# B&R Automation Studio project NAELD004C00R10L518F00 (part 20)

#### InputRef.var - Change By Project
```iecst
(*2019-03-25*)
(**)
(*Configuration*)
VAR
	p_eAct : REFERENCE TO UDINT;
	p_bOpsRun : REFERENCE TO BOOL;
END_VAR
(**)
VAR
	p_eStartupStat : REFERENCE TO eStartupAction;
	p_eStartupStatus : REFERENCE TO eFBStatus;
	p_sStartupStatTxt : REFERENCE TO STRING[200];
	p_eStartupStep : REFERENCE TO eStartupStep;
	p_sStartupStepTxt : REFERENCE TO STRING[80];
	p_bStartupGetConfigDone : REFERENCE TO BOOL;
	p_bStartupMismatchSetConfigDone : REFERENCE TO BOOL;
	p_bStartupUISettingsLoadDone : REFERENCE TO BOOL;
	p_bStartupRun : REFERENCE TO BOOL;
END_VAR
(**)
VAR
	p_eHWInfoStat : REFERENCE TO eHWInfoAction;
	p_eHWInfoStatus : REFERENCE TO eFBStatus;
	p_sHWInfoStatTxt : REFERENCE TO STRING[200];
	p_sHWInfoIPAddr : REFERENCE TO STRING[15];
	p_sHWInfoSubnetMask : REFERENCE TO STRING[15];
	p_udiHWInfoEthMode : REFERENCE TO UDINT;
END_VAR
(**)
VAR
	p_eTLBuzStat : REFERENCE TO eTLBuzAction;
	p_eTLBuzStatus : REFERENCE TO eFBStatus;
	p_sTLBuzStatTxt : REFERENCE TO STRING[200];
END_VAR
(**)
VAR
	p_tyAlarmCurrList : REFERENCE TO ARRAY[1..c_udiAlarmCurrMax] OF tyAlarmCurr;
	p_tyAlarmRcyList : REFERENCE TO ARRAY[1..c_udiAlarmCurrMax] OF UDINT;
	p_tyAlarmHistoryList : REFERENCE TO ARRAY[1..c_udiAlarmHistoryMax] OF STRING[200];
	p_bAlarmWarning : REFERENCE TO BOOL;
	p_bAlarmErr : REFERENCE TO BOOL;
	p_bAlarmInfo : REFERENCE TO BOOL;
	p_bAlarmInfoLF : REFERENCE TO BOOL;
	p_sAlarmInfoMsg : REFERENCE TO STRING[200];
END_VAR
(**)
VAR
	p_eRstErrStat : REFERENCE TO eRstErrAction;
	p_eRstErrStatus : REFERENCE TO eFBStatus;
	p_sRstErrStatTxt : REFERENCE TO STRING[200];
END_VAR
(**)
VAR
	p_eProdRcpStat : REFERENCE TO eProdRcpAction;
	p_eProdRcpStatus : REFERENCE TO eFBStatus;
	p_sProdRcpStatTxt : REFERENCE TO STRING[200];
	p_tyProdRcpFilterList : REFERENCE TO ARRAY[1..c_udiProdRcpMax] OF tyProdRcpParam;
	p_tyProdRcpSortedList : REFERENCE TO ARRAY[1..c_udiProdRcpMax] OF tyProdRcpParam;
	p_tyProdRcpCurrList : REFERENCE TO ARRAY[1..c_udiProdRcpMax] OF tyProdRcpParam;
	p_tyProdRcpCurrRcp0 : REFERENCE TO tyProdRcpParam;
	p_tyProdRcpCurrRcp1 : REFERENCE TO tyProdRcpParam;
	p_tyProdRcpCurrRcp2 : REFERENCE TO tyProdRcpParam;
	p_tyProdRcpInfoOut : REFERENCE TO tyProdRcpParam;
	p_bProdRcpNmEmpty : REFERENCE TO BOOL;
	p_bProdRcpListFull : REFERENCE TO BOOL;
	p_bProdRcpNmNotExist : REFERENCE TO BOOL;
END_VAR
(**)
VAR
	p_eMpProdRcpStat : REFERENCE TO eMpProdRcpAction;
	p_eMpProdRcpStatus : REFERENCE TO eFBStatus;
END_VAR
(**)
VAR
	p_eMagRcpStat : REFERENCE TO eMagRcpAction;
	p_eMagRcpStatus : REFERENCE TO eFBStatus;
	p_sMagRcpStatTxt : REFERENCE TO STRING[200];
	p_tyMagRcpFilterList : REFERENCE TO ARRAY[1..c_udiMagRcpMax] OF tyMagRcpParam;
	p_tyMagRcpSortedList : REFERENCE TO ARRAY[1..c_udiProdRcpMax] OF tyMagRcpParam;
	p_tyMagRcpCurrList : REFERENCE TO ARRAY[1..c_udiMagRcpMax] OF tyMagRcpParam;
	p_tyMagRcpInfoOut : REFERENCE TO tyMagRcpParam;
	p_tyMagRcpCurrRcp : REFERENCE TO tyMagRcpParam;
	p_bMagRcpNmEmpty : REFERENCE TO BOOL;
	p_bMagRcpListFull : REFERENCE TO BOOL;
	p_bMagRcpNmNotExist : REFERENCE TO BOOL;
END_VAR
(**)
VAR
	p_eMagRcpStat1 : REFERENCE TO eMagRcpAction;
	p_eMagRcpStatus1 : REFERENCE TO eFBStatus;
	p_sMagRcpStatTxt1 : REFERENCE TO STRING[200];
	p_tyMagRcpFilterList1 : REFERENCE TO ARRAY[1..c_udiMagRcpMax] OF tyMagRcpParam;
	p_tyMagRcpSortedList1 : REFERENCE TO ARRAY[1..c_udiProdRcpMax] OF tyMagRcpParam;
	p_tyMagRcpCurrList1 : REFERENCE TO ARRAY[1..c_udiMagRcpMax] OF tyMagRcpParam;
	p_tyMagRcpInfoOut1 : REFERENCE TO tyMagRcpParam;
	p_tyMagRcpCurrRcp1 : REFERENCE TO tyMagRcpParam;
	p_bMagRcpNmEmpty1 : REFERENCE TO BOOL;
	p_bMagRcpListFull1 : REFERENCE TO BOOL;
	p_bMagRcpNmNotExist1 : REFERENCE TO BOOL;
	p_diMagRcp1TravPos : REFERENCE TO DINT;
	p_diMagRcp2TravPos : REFERENCE TO DINT;
	p_diMagRcp3TravPos : REFERENCE TO DINT;
END_VAR
(**)
VAR
	p_eMcParamStat : REFERENCE TO eMcParamAction;
	p_eMcParamStatus : REFERENCE TO eFBStatus;
	p_sMcParamStatTxt : REFERENCE TO STRING[200];
	p_tyMcParamCurr : REFERENCE TO tyMcParam;
END_VAR
(**)
VAR
	p_tyNtParamCurr : REFERENCE TO tyNtParam;
END_VAR
(**)
VAR
	p_eUsrMgmtStat : REFERENCE TO eUsrMgmtAction;
	p_eUsrMgmtStatus : REFERENCE TO eFBStatus;
	p_sUsrMgmtStatTxt : REFERENCE TO STRING[200];
	p_tyUsrMgmtCurrUsr : REFERENCE TO tyUsrMgmtParam;
	p_tyUsrMgmtCurrAccessRgt : REFERENCE TO tyUsrMgmtAccessRight;
	p_tyUsrMgmtAllList : REFERENCE TO ARRAY[1..c_udiUsrMgmtMax] OF tyUsrMgmtParam;
	p_tyUsrMgmtLv2List : REFERENCE TO ARRAY[1..c_udiUsrMgmtMax] OF tyUsrMgmtParam;
	p_tyUsrMgmtLv3List : REFERENCE TO ARRAY[1..c_udiUsrMgmtMax] OF tyUsrMgmtParam;
	p_tyUsrMgmtAdminList : REFERENCE TO ARRAY[1..c_udiUsrMgmtMax] OF tyUsrMgmtParam;
	p_bUsrMgmtNmEmpty : REFERENCE TO BOOL;
	p_bUsrMgmtListFull : REFERENCE TO BOOL;
	p_bUsrMgmtNmExist : REFERENCE TO BOOL;
	p_bUsrMgmtNmNotExist : REFERENCE TO BOOL;
	p_bUsrMgmtLastAdmin : REFERENCE TO BOOL;
	p_bUsrMgmtLoginSuccess : REFERENCE TO BOOL;
	p_bUsrMgmtPwMismatch : REFERENCE TO BOOL;
	p_bUsrMgmtUnableDelete : REFERENCE TO BOOL;
	p_tyUsrMgmtFullData : REFERENCE TO tyUsrMgmtFullDat;
END_VAR
(**)
VAR
	p_eBuffer1Stat : REFERENCE TO eBufferAction;
	p_eBuffer1Status : REFERENCE TO eFBStatus;
	p_sBuffer1StatTxt : REFERENCE TO STRING[200];
	p_tyBuffer1DispBffr : REFERENCE TO tyDispBffr;
	p_tyBuffer1BffrStat : REFERENCE TO tyBffrStat;
	p_bBuffer1MagPresent : REFERENCE TO BOOL;
	p_bBuffer1MagRemoved : REFERENCE TO BOOL;
END_VAR
(**)
VAR
	p_eBuffer2Stat : REFERENCE TO eBufferAction;
	p_eBuffer2Status : REFERENCE TO eFBStatus;
	p_sBuffer2StatTxt : REFERENCE TO STRING[200];
	p_tyBuffer2DispBffr : REFERENCE TO tyDispBffr;
	p_tyBuffer2BffrStat : REFERENCE TO tyBffrStat;
	p_bBuffer2MagPresent : REFERENCE TO BOOL;
	p_bBuffer2MagRemoved : REFERENCE TO BOOL;
END_VAR
(**)
VAR
	p_eBuffer3Stat : REFERENCE TO eBufferAction;
	p_eBuffer3Status : REFERENCE TO eFBStatus;
	p_sBuffer3StatTxt : REFERENCE TO STRING[200];
	p_tyBuffer3DispBffr : REFERENCE TO tyDispBffr;
	p_tyBuffer3BffrStat : REFERENCE TO tyBffrStat;
	p_bBuffer3MagPresent : REFERENCE TO BOOL;
	p_bBuffer3MagRemoved : REFERENCE TO BOOL;
END_VAR
(**)
VAR
	p_eBuffer4Stat : REFERENCE TO eBufferAction;
	p_eBuffer4Status : REFERENCE TO eFBStatus;
	p_sBuffer4StatTxt : REFERENCE TO STRING[200];
	p_tyBuffer4DispBffr : REFERENCE TO tyDispBffr;
	p_tyBuffer4BffrStat : REFERENCE TO tyBffrStat;
	p_bBuffer4MagPresent : REFERENCE TO BOOL;
	p_bBuffer4MagRemoved : REFERENCE TO BOOL;
END_VAR
(**)
VAR
	p_eDSSMEMAAStat : REFERENCE TO eSMEMAAction;
	p_eDSSMEMAAStatus : REFERENCE TO eFBStatus;
	p_sDSSMEMAAStatTxt : REFERENCE TO STRING[200];
	p_bDSSMEMAAUSRdy : REFERENCE TO BOOL;
	p_bDSSMEMAAUSGdBrdRdy : REFERENCE TO BOOL;
	p_bDSSMEMAADSRdy : REFERENCE TO BOOL;
END_VAR
(**)
VAR
	p_eDSSMEMABStat : REFERENCE TO eSMEMAAction;
	p_eDSSMEMABStatus : REFERENCE TO eFBStatus;
	p_sDSSMEMABStatTxt : REFERENCE TO STRING[200];
	p_bDSSMEMABUSRdy : REFERENCE TO BOOL;
	p_bDSSMEMABUSGdBrdRdy : REFERENCE TO BOOL;
	p_bDSSMEMABDSRdy : REFERENCE TO BOOL;
END_VAR
(**)
VAR
	p_eInShutterStat : REFERENCE TO ePneuAction;
	p_eInShutterStatus : REFERENCE TO eFBStatus;
	p_sInShutterStatTxt : REFERENCE TO STRING[200];
	p_bInShutterExtCtrl : REFERENCE TO BOOL;
	p_bInShutterRetCtrl : REFERENCE TO BOOL;
	p_bInShutterTwoCtrlOut : REFERENCE TO BOOL;
	p_bInShutterExtended : REFERENCE TO BOOL;
	p_bInShutterRetracted : REFERENCE TO BOOL;
END_VAR
(**)
VAR
	p_eInShutterStat2 : REFERENCE TO ePneuAction;
	p_eInShutterStatus2 : REFERENCE TO eFBStatus;
	p_sInShutterStatTxt2 : REFERENCE TO STRING[200];
	p_bInShutterExtCtrl2 : REFERENCE TO BOOL;
	p_bInShutterRetCtrl2 : REFERENCE TO BOOL;
	p_bInShutterTwoCtrlOut2 : REFERENCE TO BOOL;
	p_bInShutterExtended2 : REFERENCE TO BOOL;
	p_bInShutterRetracted2 : REFERENCE TO BOOL;
END_VAR
(**)
VAR
	p_eInShutterStat3 : REFERENCE TO ePneuAction;
	p_eInShutterStatus3 : REFERENCE TO eFBStatus;
	p_sInShutterStatTxt3 : REFERENCE TO STRING[200];
	p_bInShutterExtCtrl3 : REFERENCE TO BOOL;
	p_bInShutterRetCtrl3 : REFERENCE TO BOOL;
	p_bInShutterTwoCtrlOut3 : REFERENCE TO BOOL;
	p_bInShutterExtended3 : REFERENCE TO BOOL;
	p_bInShutterRetracted3 : REFERENCE TO BOOL;
END_VAR
(**)
VAR
	p_eOutShutterStat : REFERENCE TO ePneuAction;
	p_eOutShutterStatus : REFERENCE TO eFBStatus;
	p_sOutShutterStatTxt : REFERENCE TO STRING[200];
	p_bOutShutterExtCtrl : REFERENCE TO BOOL;
	p_bOutShutterRetCtrl : REFERENCE TO BOOL;
	p_bOutShutterTwoCtrlOut : REFERENCE TO BOOL;
	p_bOutShutterExtended : REFERENCE TO BOOL;
	p_bOutShutterRetracted : REFERENCE TO BOOL;
END_VAR
(**)
VAR
	p_eOutShutterStat2 : REFERENCE TO ePneuAction;
	p_eOutShutterStatus2 : REFERENCE TO eFBStatus;
	p_sOutShutterStatTxt2 : REFERENCE TO STRING[200];
	p_bOutShutterExtCtrl2 : REFERENCE TO BOOL;
	p_bOutShutterRetCtrl2 : REFERENCE TO BOOL;
	p_bOutShutterTwoCtrlOut2 : REFERENCE TO BOOL;
	p_bOutShutterExtended2 : REFERENCE TO BOOL;
	p_bOutShutterRetracted2 : REFERENCE TO BOOL;
END_VAR
(**)
VAR
	p_eSelClamp1Stat : REFERENCE TO ePneuAction;
	p_eSelClamp1Status : REFERENCE TO eFBStatus;
	p_sSelClamp1StatTxt : REFERENCE TO STRING[200];
	p_bSelClamp1ExtCtrl : REFERENCE TO BOOL;
	p_bSelClamp1RetCtrl : REFERENCE TO BOOL;
	p_bSelClamp1TwoCtrlOut : REFERENCE TO BOOL;
	p_bSelClamp1Extended : REFERENCE TO BOOL;
	p_bSelClamp1Retracted : REFERENCE TO BOOL;
END_VAR
(**)
VAR
	p_eSelClamp2Stat : REFERENCE TO ePneuAction;
	p_eSelClamp2Status : REFERENCE TO eFBStatus;
	p_sSelClamp2StatTxt : REFERENCE TO STRING[200];
	p_bSelClamp2ExtCtrl : REFERENCE TO BOOL;
	p_bSelClamp2RetCtrl : REFERENCE TO BOOL;
	p_bSelClamp2TwoCtrlOut : REFERENCE TO BOOL;
	p_bSelClamp2Extended : REFERENCE TO BOOL;
	p_bSelClamp2Retracted : REFERENCE TO BOOL;
END_VAR
(**)
VAR
	p_eSelClamp3Stat : REFERENCE TO ePneuAction;
	p_eSelClamp3Status : REFERENCE TO eFBStatus;
	p_sSelClamp3StatTxt : REFERENCE TO STRING[200];
	p_bSelClamp3ExtCtrl : REFERENCE TO BOOL;
	p_bSelClamp3RetCtrl : REFERENCE TO BOOL;
	p_bSelClamp3TwoCtrlOut : REFERENCE TO BOOL;
	p_bSelClamp3Extended : REFERENCE TO BOOL;
	p_bSelClamp3Retracted : REFERENCE TO BOOL;
END_VAR
(**)
VAR
	p_eSelClamp4Stat : REFERENCE TO ePneuAction;
	p_eSelClamp4Status : REFERENCE TO eFBStatus;
	p_sSelClamp4StatTxt : REFERENCE TO STRING[200];
	p_bSelClamp4ExtCtrl : REFERENCE TO BOOL;
	p_bSelClamp4RetCtrl : REFERENCE TO BOOL;
	p_bSelClamp4TwoCtrlOut : REFERENCE TO BOOL;
	p_bSelClamp4Extended : REFERENCE TO BOOL;
	p_bSelClamp4Retracted : REFERENCE TO BOOL;
END_VAR
(**)
VAR
	p_ePullerStat : REFERENCE TO ePneuAction;
	p_ePullerStatus : REFERENCE TO eFBStatus;
	p_sPullerStatTxt : REFERENCE TO STRING[200];
	p_bPullerExtCtrl : REFERENCE TO BOOL;
	p_bPullerRetCtrl : REFERENCE TO BOOL;
	p_bPullerTwoCtrlOut : REFERENCE TO BOOL;
	p_bPullerExtended : REFERENCE TO BOOL;
	p_bPullerRetracted : REFERENCE TO BOOL;
END_VAR
(**)
VAR
	p_ePullConvStat : REFERENCE TO eConvAction;
	p_ePullConvStatus : REFERENCE TO eFBStatus;
	p_sPullConvStatTxt : REFERENCE TO STRING[200];
	p_bPullConvHvBrd : REFERENCE TO BOOL;
	p_bPullConvGdBrd : REFERENCE TO BOOL;
	p_bPullConvMtrSigOnOrLToR : REFERENCE TO BOOL;
	p_bPullConvMtrDirOrRToL : REFERENCE TO BOOL;
	p_bPullConvPullerExtCtrl : REFERENCE TO BOOL;
	p_bPullConvPullerRetCtrl : REFERENCE TO BOOL;
	p_bPullConvPullerTwoOutputCtrl : REFERENCE TO BOOL;
	p_bPullConvRotRemoteCtrl : REFERENCE TO BOOL;
	p_bPullConvRotTwoOutputCtrl : REFERENCE TO BOOL;
END_VAR
(**)
VAR
	p_eMagConv2Clp1Stat : REFERENCE TO eMagConv2ClpAction;
	p_eMagConv2Clp1Status : REFERENCE TO eFBStatus;
	p_sMagConv2Clp1StatTxt : REFERENCE TO STRING[200];
	p_bMagConv2Clp1HvMag : REFERENCE TO BOOL;
	p_bMagConv2Clp1MtrSigOnOrLToR : REFERENCE TO BOOL;
	p_bMagConv2Clp1MtrDirOrRToL : REFERENCE TO BOOL;
	p_bMagConv2Clp1ClprFixClampCtrl : REFERENCE TO BOOL;
	p_bMagConv2Clp1ClprRmtClampCtrl : REFERENCE TO BOOL;
	p_bMagConv2Clp1ClprTwoOutputCtrl : REFERENCE TO BOOL;
END_VAR
(**)
VAR
	p_eMagConv2Clp2Stat : REFERENCE TO eMagConv2ClpAction;
	p_eMagConv2Clp2Status : REFERENCE TO eFBStatus;
	p_sMagConv2Clp2StatTxt : REFERENCE TO STRING[200];
	p_bMagConv2Clp2HvMag : REFERENCE TO BOOL;
	p_bMagConv2Clp2MtrSigOnOrLToR : REFERENCE TO BOOL;
	p_bMagConv2Clp2MtrDirOrRToL : REFERENCE TO BOOL;
	p_bMagConv2Clp2ClprFixClampCtrl : REFERENCE TO BOOL;
	p_bMagConv2Clp2ClprRmtClampCtrl : REFERENCE TO BOOL;
	p_bMagConv2Clp2ClprTwoOutputCtrl : REFERENCE TO BOOL;
END_VAR
(**)
VAR
	p_eMagConv2Clp3Stat : REFERENCE TO eMagConv2ClpAction;
	p_eMagConv2Clp3Status : REFERENCE TO eFBStatus;
	p_sMagConv2Clp3StatTxt : REFERENCE TO STRING[200];
	p_bMagConv2Clp3HvMag : REFERENCE TO BOOL;
	p_bMagConv2Clp3MtrSigOnOrLToR : REFERENCE TO BOOL;
	p_bMagConv2Clp3MtrDirOrRToL : REFERENCE TO BOOL;
	p_bMagConv2Clp3ClprFixClampCtrl : REFERENCE TO BOOL;
	p_bMagConv2Clp3ClprRmtClampCtrl : REFERENCE TO BOOL;
	p_bMagConv2Clp3ClprTwoOutputCtrl : REFERENCE TO BOOL;
END_VAR
(**)
VAR
	p_eMagConv2Clp4Stat : REFERENCE TO eMagConv2ClpAction;
	p_eMagConv2Clp4Status : REFERENCE TO eFBStatus;
	p_sMagConv2Clp4StatTxt : REFERENCE TO STRING[200];
	p_bMagConv2Clp4HvMag : REFERENCE TO BOOL;
	p_bMagConv2Clp4MtrSigOnOrLToR : REFERENCE TO BOOL;
	p_bMagConv2Clp4MtrDirOrRToL : REFERENCE TO BOOL;
	p_bMagConv2Clp4ClprFixClampCtrl : REFERENCE TO BOOL;
	p_bMagConv2Clp4ClprRmtClampCtrl : REFERENCE TO BOOL;
	p_bMagConv2Clp4ClprTwoOutputCtrl : REFERENCE TO BOOL;
END_VAR
(**)
VAR
	p_eAWPushOrPullerStat : REFERENCE TO eAWAction;
	p_eAWPushOrPullerStatus : REFERENCE TO eFBStatus;
	p_sAWPushOrPullerStatTxt : REFERENCE TO STRING[200];
	p_udiAWPushOrPullerAxisErrID : REFERENCE TO UDINT;
	p_bAWPushOrPullerAxisErr : REFERENCE TO BOOL;
	p_bAWPushOrPullerPwrOn : REFERENCE TO BOOL;
	p_bAWPushOrPullerIsHomed : REFERENCE TO BOOL;
	p_diAWPushOrPullerActualPos : REFERENCE TO DINT;
	p_bAWPushOrPullerFwdLmtSen : REFERENCE TO BOOL;
	p_bAWPushOrPullerRevLmtSen : REFERENCE TO BOOL;
	p_sAWPushOrPullerAxisErrTxt : REFERENCE TO STRING[80];
	p_bAWPushOrPullerJogging : REFERENCE TO BOOL;
	p_bAWPushOrPullerOpenSen : REFERENCE TO BOOL;
	p_bAWPushOrPullerCloseSen : REFERENCE TO BOOL;
	p_bAWPushOrPullerPrep : REFERENCE TO BOOL;
END_VAR
(**)
VAR
	p_eAWOpenStat : REFERENCE TO eAWAction;
	p_eAWOpenStatus : REFERENCE TO eFBStatus;
	p_sAWOpenStatTxt : REFERENCE TO STRING[200];
	p_udiAWOpenAxisErrID : REFERENCE TO UDINT;
	p_bAWOpenAxisErr : REFERENCE TO BOOL;
	p_bAWOpenPwrOn : REFERENCE TO BOOL;
	p_bAWOpenIsHomed : REFERENCE TO BOOL;
	p_diAWOpenActualPos : REFERENCE TO DINT;
	p_bAWOpenFwdLmtSen : REFERENCE TO BOOL;
	p_bAWOpenRevLmtSen : REFERENCE TO BOOL;
	p_bAWOpenWidthPosDiff : REFERENCE TO BOOL;
	p_sAWOpenAxisErrTxt : REFERENCE TO STRING[80];
	p_bAWOpenJogging : REFERENCE TO BOOL;
	p_bAWOpenOpenSen : REFERENCE TO BOOL;
	p_bAWOpenCloseSen : REFERENCE TO BOOL;
END_VAR
(**)
VAR
	p_eLifterBtmStat : REFERENCE TO eLifterAction;
	p_eLifterBtmStatus : REFERENCE TO eFBStatus;
	p_sLifterBtmStatTxt : REFERENCE TO STRING[200];
	p_bLifterBtmPwrOn : REFERENCE TO BOOL;
	p_bLifterBtmIsHomed : REFERENCE TO BOOL;
	p_bLifterBtmPosDiff : REFERENCE TO BOOL;
	p_bLifterBtmAxisErr : REFERENCE TO BOOL;
	p_udiLifterBtmAxisErrID : REFERENCE TO UDINT;
	p_sLifterBtmAxisErrTxt : REFERENCE TO STRING[80];
	p_bLifterBtmFwdLmtSen : REFERENCE TO BOOL;
	p_bLifterBtmRevLmtSen : REFERENCE TO BOOL;
	p_diLifterBtmActualPos : REFERENCE TO DINT;
	p_bLifterBtmJogging : REFERENCE TO BOOL;
	p_diLifterBtmCurrSltA : REFERENCE TO DINT;
	p_diLifterBtmCurrSltB : REFERENCE TO DINT;
	p_diLifterBtmCurrSltC : REFERENCE TO DINT;
	p_bLifterBtmUpSen : REFERENCE TO BOOL;
	p_bLifterBtmDownSen : REFERENCE TO BOOL;
	p_bLifterBtmSltAPosDiff : REFERENCE TO BOOL;
END_VAR
(**)
VAR
	p_eTravStat : REFERENCE TO eTravAction;
	p_eTravStatus : REFERENCE TO eFBStatus;
	p_sTravStatTxt : REFERENCE TO STRING[200];
	p_bTravPwrOn : REFERENCE TO BOOL;
	p_bTravIsHomed : REFERENCE TO BOOL;
	p_bTravPosDiff : REFERENCE TO BOOL;
	p_bTravAxisErr : REFERENCE TO BOOL;
	p_udiTravAxisErrID : REFERENCE TO UDINT;
	p_sTravAxisErrTxt : REFERENCE TO STRING[80];
	p_bTravFwdLmtSen : REFERENCE TO BOOL;
	p_bTravRevLmtSen : REFERENCE TO BOOL;
	p_diTravActualPos : REFERENCE TO DINT;
	p_bTravJogging : REFERENCE TO BOOL;
	p_bTravFrontSen : REFERENCE TO BOOL;
	p_bTravRearSen : REFERENCE TO BOOL;
	p_bTravAPosDiff : REFERENCE TO BOOL;
	p_bTravBPosDiff : REFERENCE TO BOOL;
	p_bTravCPosDiff : REFERENCE TO BOOL;
	p_bTravDPosDiff : REFERENCE TO BOOL;
	p_bTravEPosDiff : REFERENCE TO BOOL;
	p_bTravFPosDiff : REFERENCE TO BOOL;
	p_bTravGPosDiff : REFERENCE TO BOOL;
	p_bTravHPosDiff : REFERENCE TO BOOL;
END_VAR
(**)
VAR
	p_tyDI : REFERENCE TO tyDigitalInput;
END_VAR
(**)
VAR
	p_eDOStat : REFERENCE TO eDOAction;
	p_eDOStatus : REFERENCE TO eFBStatus;
	p_sDOStatTxt : REFERENCE TO STRING[200];
	p_tyDO : REFERENCE TO tyDigitalOutput;
END_VAR
(**)
VAR
	p_tyDTMagToAGV1 : REFERENCE TO tyTagDTMagToAGV;
	p_tyDTMagToAGV2 : REFERENCE TO tyTagDTMagToAGV;
	p_tyDTMagToAGV3 : REFERENCE TO tyTagDTMagToAGV;
	p_tyDTMagToAGV4 : REFERENCE TO tyTagDTMagToAGV;
	p_tyAGVToDTMag : REFERENCE TO tyTagAGVToDTMag;
	p_bAGVOnline : REFERENCE TO BOOL;
	p_bMachineOnline : REFERENCE TO BOOL;
	p_bAGVSimulationOn : REFERENCE TO BOOL;
	p_tyDTMagToAGV : REFERENCE TO tyTagDTMagToAGV;
	p_tyTagToMes : REFERENCE TO tyStatToMES;
	p_tyTagFromMes : REFERENCE TO tyStatFromMES;
END_VAR
(**)
VAR
	p_eHermesStat : REFERENCE TO eHermesAction;
	p_eHermesStatus : REFERENCE TO eFBStatus;
	p_tyHermesConfiguration : REFERENCE TO tyHermesConfiguration;
	p_bRmtUpdateUIData : REFERENCE TO BOOL;
	p_bSvyUpdateUIData : REFERENCE TO BOOL;
	p_bRcvBoardInfoOk : REFERENCE TO BOOL;
	p_bRcvBoardInfoIncompl : REFERENCE TO BOOL;
	p_bTransportFinished : REFERENCE TO BOOL;
	p_bWaitDecision : REFERENCE TO BOOL;
	p_sWorkOrderId : REFERENCE TO STRING[80];
END_VAR
(**)
VAR
	p_eDSHermesAStat : REFERENCE TO eHermesAction;
	p_eDSHermesAStatus : REFERENCE TO eFBStatus;
	p_sDSHermesAStatTxt : REFERENCE TO STRING[200];
	p_bDSHermesAUSRdy : REFERENCE TO BOOL;
	p_bDSHermesADSRdy : REFERENCE TO BOOL;
	p_bDSHermesAUSGdRdy : REFERENCE TO BOOL;
	p_bDSHermesADSGdRdy : REFERENCE TO BOOL;
	p_bDSHermesAConnected : REFERENCE TO BOOL;
END_VAR
(**)
VAR
	p_eDSHermesBStat : REFERENCE TO eHermesAction;
	p_eDSHermesBStatus : REFERENCE TO eFBStatus;
	p_sDSHermesBStatTxt : REFERENCE TO STRING[200];
	p_bDSHermesBUSRdy : REFERENCE TO BOOL;
	p_bDSHermesBDSRdy : REFERENCE TO BOOL;
	p_bDSHermesBUSGdRdy : REFERENCE TO BOOL;
	p_bDSHermesBDSGdRdy : REFERENCE TO BOOL;
	p_bDSHermesBConnected : REFERENCE TO BOOL;
END_VAR
(**)
VAR
	p_eLFLeaderStat : REFERENCE TO eLFAction;
	p_eLFLeaderStatus : REFERENCE TO eFBStatus;
	p_tyLFLeaderFollowerInfo : REFERENCE TO ARRAY[1..c_diLFClntNum] OF tyLFFollowerInfo;
	p_tyLFLeaderFollowerToLeaderTag : REFERENCE TO ARRAY[1..c_diLFClntNum] OF tyLFFollowerToLeaderTag;
END_VAR
(**)
VAR
	p_bLFFollowerProdAccDataMnl : REFERENCE TO BOOL;
	p_bLFFollowerLdrSeqCtrlInActive : REFERENCE TO BOOL;
	p_bLFFollowerUSAllow : REFERENCE TO BOOL;
	p_bLFFollowerDSAllow : REFERENCE TO BOOL;
END_VAR
(**)
VAR
	p_bLCSLFAccDataMnl : REFERENCE TO BOOL;
END_VAR
(**)
VAR
	p_eOpsStat : REFERENCE TO eOperationsAction;
	p_eOpsStatus : REFERENCE TO eFBStatus;
	p_sOpsStatTxt : REFERENCE TO STRING[200];
	p_eOpsOpsStatus : REFERENCE TO eOperationsStatus;
	p_bOpsStatusRun : REFERENCE TO BOOL;
	p_bOpsStatusStop : REFERENCE TO BOOL;
	p_bOpsStatusCycleStop : REFERENCE TO BOOL;
	p_bOpsStatusStep : REFERENCE TO BOOL;
END_VAR
(**)
VAR
	p_sOpsTravLifLDStepTxt : REFERENCE TO STRING[80];
	p_sOpsMagLD1StepTxt : REFERENCE TO STRING[80];
	p_sOpsMagLD2StepTxt : REFERENCE TO STRING[80];
	p_sOpsMagLD3StepTxt : REFERENCE TO STRING[80];
	p_sOpsMagLD4StepTxt : REFERENCE TO STRING[80];
	p_sOpsMagConvLD1StepTxt : REFERENCE TO STRING[80];
	p_sOpsMagConvLD2StepTxt : REFERENCE TO STRING[80];
	p_sOpsMagConvLD3StepTxt : REFERENCE TO STRING[80];
	p_sOpsMagConvLD4StepTxt : REFERENCE TO STRING[80];
END_VAR
(**)
VAR
	p_bOpsTravLifLDInitConv : REFERENCE TO BOOL;
	p_bOpsTravLifLDAWPosDiff : REFERENCE TO BOOL;
	p_bOpsTravLifLDExitBrd : REFERENCE TO BOOL;
	p_eOpsTravLifPosGo : REFERENCE TO eTravLifLDPos;
	p_bOpsTravLifStandby : REFERENCE TO BOOL;
	p_bOpsMagConvLD1InitDone : REFERENCE TO BOOL;
	p_bOpsMagConvLD2InitDone : REFERENCE TO BOOL;
	p_bOpsMagConvLD3InitDone : REFERENCE TO BOOL;
	p_bOpsMagConvLD4InitDone : REFERENCE TO BOOL;
	p_bOpsMagConvLD1MagExitedWait : REFERENCE TO BOOL;
	p_bOpsMagConvLD2MagExitedWait : REFERENCE TO BOOL;
	p_bOpsMagConvLD3MagExitedWait : REFERENCE TO BOOL;
	p_bOpsMagConvLD4MagExitedWait : REFERENCE TO BOOL;
	p_bOpsMagConvLD1NewMagAllw : REFERENCE TO BOOL;
	p_bOpsMagConvLD2NewMagAllw : REFERENCE TO BOOL;
	p_bOpsMagConvLD3NewMagAllw : REFERENCE TO BOOL;
	p_bOpsMagConvLD4NewMagAllw : REFERENCE TO BOOL;
	p_bOpsMagConvLD1RlsMagAllw : REFERENCE TO BOOL;
	p_bOpsMagConvLD2RlsMagAllw : REFERENCE TO BOOL;
	p_bOpsMagConvLD3RlsMagAllw : REFERENCE TO BOOL;
	p_bOpsMagConvLD4RlsMagAllw : REFERENCE TO BOOL;
	p_bOpsMagConvLD1RlsMagUmask : REFERENCE TO BOOL;
	p_bOpsMagConvLD2RlsMagUmask : REFERENCE TO BOOL;
	p_bOpsMagConvLD3RlsMagUmask : REFERENCE TO BOOL;
	p_bOpsMagConvLD1ExtMes : REFERENCE TO BOOL;
	p_bOpsMagConvLD2ExtMes : REFERENCE TO BOOL;
	p_bOpsMagConvLD3ExtMes : REFERENCE TO BOOL;
	p_bOpsMagConvLD1HModChgDone : REFERENCE TO BOOL;
	p_bOpsMagConvLD2HModChgDone : REFERENCE TO BOOL;
	p_bOpsMagConvLD3HModChgDone : REFERENCE TO BOOL;
END_VAR
(**)
VAR
	p_bOpsLifMagLDUnloading : REFERENCE TO BOOL;
	p_sOpsLifMagLDStepTxt : REFERENCE TO STRING[80];
END_VAR
(**)
VAR
	p_eSimuStat : REFERENCE TO eSimulationsAction;
	p_eSimuStatus : REFERENCE TO eFBStatus;
	p_eSimuSimuStatus : REFERENCE TO eSimulationsStatus;
	p_bSimuStatusRun : REFERENCE TO BOOL;
	p_bSimuStatusStop : REFERENCE TO BOOL;
	p_bSimuStatusCycleStop : REFERENCE TO BOOL;
	p_bSimuStatusStep : REFERENCE TO BOOL;
	p_sNtParamJobNo : REFERENCE TO STRING[30];
	p_usiNtParamNtAddr : REFERENCE TO USINT;
	p_eNtParamStat : REFERENCE TO eNtParamAction;
	p_eNtParamStatus : REFERENCE TO eFBStatus;
	p_diNtParamLifterAutoSpd : REFERENCE TO DINT;
	p_diNtParamTravAutoSpd : REFERENCE TO DINT;
END_VAR
(**)
VAR
	p_eUSBRdrStat : REFERENCE TO eUSBRdrAction;
	p_eUSBRdrStatus : REFERENCE TO eFBStatus;
	p_sUSBRdrBarcodeOut : REFERENCE TO STRING[255];
	p_bUSBDisconnected : REFERENCE TO BOOL;
END_VAR
(**)
VAR
	p_eFrmStat : REFERENCE TO eFrmAction;
	p_eFrmStatus : REFERENCE TO eFBStatus;
	p_sFrmFullMsgRd : REFERENCE TO STRING[15];
	p_sFrmMsgRd : REFERENCE TO STRING[15];
	p_bFrmMsgRdValid : REFERENCE TO BOOL;
	p_uiFrmMsgRdLen : REFERENCE TO UINT;
END_VAR
(**)
VAR
	p_eMtrPshrStat : REFERENCE TO eMtrPshrAction;
	p_eMtrPshrStatus : REFERENCE TO eFBStatus;
	p_sMtrPshrStatTxt : REFERENCE TO STRING[200];
END_VAR
(**)
VAR
	p_eMag1SafetyBarStat : REFERENCE TO ePneuAction;
	p_eMag1SafetyBarStatus : REFERENCE TO eFBStatus;
	p_sMag1SafetyBarStatTxt : REFERENCE TO STRING[200];
	p_bMag1SafetyBarExtCtrl : REFERENCE TO BOOL;
	p_bMag1SafetyBarRetCtrl : REFERENCE TO BOOL;
	p_bMag1SafetyBarTwoCtrlOut : REFERENCE TO BOOL;
	p_bMag1SafetyBarExtended : REFERENCE TO BOOL;
	p_bMag1SafetyBarRetracted : REFERENCE TO BOOL;
END_VAR
(**)
VAR
	p_eMag2SafetyBarStat : REFERENCE TO ePneuAction;
	p_eMag2SafetyBarStatus : REFERENCE TO eFBStatus;
	p_sMag2SafetyBarStatTxt : REFERENCE TO STRING[200];
	p_bMag2SafetyBarExtCtrl : REFERENCE TO BOOL;
	p_bMag2SafetyBarRetCtrl : REFERENCE TO BOOL;
	p_bMag2SafetyBarTwoCtrlOut : REFERENCE TO BOOL;
	p_bMag2SafetyBarExtended : REFERENCE TO BOOL;
	p_bMag2SafetyBarRetracted : REFERENCE TO BOOL;
END_VAR
(**)
VAR
	p_eMag3SafetyBarStat : REFERENCE TO ePneuAction;
	p_eMag3SafetyBarStatus : REFERENCE TO eFBStatus;
	p_sMag3SafetyBarStatTxt : REFERENCE TO STRING[200];
	p_bMag3SafetyBarExtCtrl : REFERENCE TO BOOL;
	p_bMag3SafetyBarRetCtrl : REFERENCE TO BOOL;
	p_bMag3SafetyBarTwoCtrlOut : REFERENCE TO BOOL;
	p_bMag3SafetyBarExtended : REFERENCE TO BOOL;
	p_bMag3SafetyBarRetracted : REFERENCE TO BOOL;
END_VAR
(**)
VAR
	p_eTrolleyLckStat : REFERENCE TO ePneuAction;
	p_eTrolleyLckStatus : REFERENCE TO eFBStatus;
	p_sTrolleyLckStatTxt : REFERENCE TO STRING[200];
	p_bTrolleyLckExtCtrl : REFERENCE TO BOOL;
	p_bTrolleyLckRetCtrl : REFERENCE TO BOOL;
	p_bTrolleyLckTwoCtrlOut : REFERENCE TO BOOL;
	p_bTrolleyLckExtended : REFERENCE TO BOOL;
	p_bTrolleyLckRetracted : REFERENCE TO BOOL;
END_VAR
(**)
VAR
	p_eTrolleyLckStat2 : REFERENCE TO ePneuAction;
	p_eTrolleyLckStatus2 : REFERENCE TO eFBStatus;
	p_sTrolleyLckStatTxt2 : REFERENCE TO STRING[200];
	p_bTrolleyLckExtCtrl2 : REFERENCE TO BOOL;
	p_bTrolleyLckRetCtrl2 : REFERENCE TO BOOL;
	p_bTrolleyLckTwoCtrlOut2 : REFERENCE TO BOOL;
	p_bTrolleyLckExtended2 : REFERENCE TO BOOL;
	p_bTrolleyLckRetracted2 : REFERENCE TO BOOL;
END_VAR
(**)
VAR
	p_diNtParamPullerHeightInMM : REFERENCE TO DINT;
END_VAR
(**)
VAR
	p_ePPStat : REFERENCE TO eTravAction;
	p_ePPStatus : REFERENCE TO eFBStatus;
	p_sPPStatTxt : REFERENCE TO STRING[200];
	p_bPPPwrOn : REFERENCE TO BOOL;
	p_bPPIsHomed : REFERENCE TO BOOL;
	p_bPPPosDiff : REFERENCE TO BOOL;
	p_bPPAxisErr : REFERENCE TO BOOL;
	p_udiPPAxisErrID : REFERENCE TO UDINT;
	p_sPPAxisErrTxt : REFERENCE TO STRING[80];
	p_bPPFwdLmtSen : REFERENCE TO BOOL;
	p_bPPRevLmtSen : REFERENCE TO BOOL;
	p_diPPActualPos : REFERENCE TO DINT;
	p_bPPJogging : REFERENCE TO BOOL;
	p_bPPExtSen : REFERENCE TO BOOL;
	p_bPPRetSen : REFERENCE TO BOOL;
	p_tyMcAlmData : REFERENCE TO tyAlmDat;
END_VAR
(*Hermes 1.3 extra*)
VAR
	p_tySendWorkOrderData : REFERENCE TO tyHermesSendWorkOrderInfo;
	p_tySvyHermesSendWorkOrderData : REFERENCE TO tyHermesSendWorkOrderInfo;
	p_tySvyHermesBypassSendWOData : REFERENCE TO tyHermesSendWorkOrderInfo;
	p_diReqLoaderWidthInUM : REFERENCE TO DINT;
	p_bQueryBypassWorkOrder : REFERENCE TO BOOL;
	p_bReplyBypassWorkOrderInfo : REFERENCE TO BOOL;
	p_bRcvWorkOrderInfo1 : REFERENCE TO BOOL;
	p_bNewIncomingBoard : REFERENCE TO BOOL;
END_VAR
(*autorcp*)
VAR
	p_diLinkAutoRcpMag1Pitch : REFERENCE TO DINT;
	p_diLinkAutoRcpMag1MinSlt : REFERENCE TO DINT;
	p_diLinkAutoRcpMag1MaxSlt : REFERENCE TO DINT;
	p_diLinkAutoRcpMag2Pitch : REFERENCE TO DINT;
	p_diLinkAutoRcpMag2MinSlt : REFERENCE TO DINT;
	p_diLinkAutoRcpMag2MaxSlt : REFERENCE TO DINT;
	p_diLinkAutoRcpMag3Pitch : REFERENCE TO DINT;
	p_diLinkAutoRcpMag3MinSlt : REFERENCE TO DINT;
	p_diLinkAutoRcpMag3MaxSlt : REFERENCE TO DINT;
	p_ausiSvyMagAccOrder : REFERENCE TO ARRAY[1..3] OF USINT;
	p_tyAutoRcpMagRcp : REFERENCE TO ARRAY[1..4] OF tyBoardProperty;
END_VAR
(**)
```

#### Local.typ - Change By Project
```iecst
(*2018-12-10*)
(**)

TYPE
	ePage :
		(
		UIP0000SSaver := 0, (*Page Screen Saver*)
		UIP0001Startup := 1, (*Page Startup*)
		UIP0002Menu := 2, (*Page Menu*)
		UIP0100Login := 100, (*Page Login*)
		UIP0200OpsGen := 200, (*Page Operation*)
		UIP0201OpsTravLifter := 201, (*Page Operation Traverser Lifter*)
		UIP0202OpsMag1 := 202, (*Page Operation Magazine 1*)
		UIP0203OpsMag2 := 203, (*Page Operation Magazine 2*)
		UIP0204OpsMag3 := 204, (*Page Operation Magazine 3*)
		UIP0205OpsAIV := 205, (*Page Operation Magazine 3*)
		UIP0206OpsMag4 := 206, (*Page Operation Magazine 3*)
		UIP0300McInfo := 300, (*Page Machine Info*)
		UIP0400ProdSel := 400, (*Page Product Selection*)
		UIP0410MagSel := 410, (*Page Magazine Selection*)
		UIP0600Alm := 600, (*Page Alarm*)
		UIP0700LFCtrl := 700, (*Page Leader Follower Control*)
		UIP0800MagInfo := 800, (*Page Magazine Info*)
		UIP0900GenIn := 900, (*Page General Input*)
		UIP0910GenOut := 910, (*Page General Output*)
		UIP0920MtrNPneuCtrl := 920, (*Page Motor And Pneumatic Control*)
		UIP0921Shutter := 921, (*Page Shutter*)
		UIP0923SafetyBar := 923, (*Page Safety Bar*)
		UIP0924TrolleyLck := 924, (*Page Safety Bar*)
		UIP0930MagConv1 := 930, (*Page Magazine Conveyor 1*)
		UIP0931MagConv2 := 931, (*Page Magazine Conveyor 2*)
		UIP0932MagConv3 := 932, (*Page Magazine Conveyor 3*)
		UIP0933PullConv := 933, (*Page Puller Conveyor*)
		UIP0934AW := 934, (*Page Auto Width*)
		UIP0935Lifter := 935, (*Page Lifter*)
		UIP0936Trav := 936, (*Page Traverser*)
		UIP0937AWPushOrPuller := 937, (*Page Pusher Auto Width*)
		UIP0939MagConv4 := 939, (*Page Magazine Conveyor 3*)
		UIP0940CommCtrl := 940, (*Page Communication Control*)
		UIP0950Simu := 950, (*Page Simulation*)
		UIP1000Lang := 1000, (*Page Language And Setup*)
		UIP1020McSetNavi := 1020, (*Page Machine Setting - Navigation*)
		UIP1021McSetGen := 1021, (*Page Machine Setting - General*)
		UIP1022McSetVComm := 1022, (*Page Machine Setting - Vertical Communication*)
		UIP1023McSetHComm := 1023, (*Page Machine Setting - Horizontal Communication*)
		UIP1024McSetAntiGap := 1024, (*Page Machine Setting - Anti Gap*)
		UIP1025McSetAIVComm := 1025, (*Page Machine Setting - AIV Communication*)
		UIP1026McSetTeach := 1026, (*Page Machine Setting - Teaching*)
		UIP1027McSetUSBSet := 1027, (*Page Machine Setting - USB*)
		UIP1028McSetRS232Set := 1028, (*Page Machine Settings RS232 Settings*)
		UIP1030MagSet := 1030, (*Page Magazine Setting*)
		UIP1031MagSetTeach := 1031, (*Page Magazine Setting - Teaching*)
		UIP1040ProdSet := 1040, (*Page Product Setting*)
		UIP1050LFSet := 1050, (*Page Leader Follower Setup*)
		UIP1080UsrMgmt := 1080, (*Page User Management*)
		UIP1081UsrMgmtUsrAccessRgt := 1081 (*Page User Management - Access Right*)
		);
	tyTable : 	STRUCT
		bSliderActive : BOOL := FALSE;
		bTableActive : BOOL := FALSE;
		sVisuNm : STRING[80] := 'Visu';
		uiSelectedRow : UINT := 1;
		uiSelectedRowOld : UINT := 1;
		uiTablePos : UINT := 1;
	END_STRUCT;
END_TYPE

(**)

TYPE
	tyUITagNm : 	STRUCT
		sWorkOrder : STRING[30];
		uiQuantities : UINT;
		diTotalBrd : DINT;
		sLogMessage : STRING[80];
		bProcess : BOOL;
	END_STRUCT;
END_TYPE
```

#### Local.var - Change By Project
```iecst
(*2019-03-25*)
(**)
(*Local Action, State & Status*)
VAR
	eAct : eUIAction := UIActIdle;
	eStat : eUIAction := UIActIdle;
	eStatus : eFBStatus := Idle;
	sStatTxt : STRING[200] := '';
	a_sStatText : ARRAY[0..50] OF STRING[200] := ['Idling','Initializing UI Page',49('')];
END_VAR
(**)
(*All General Alarm*)
VAR
	tyUIAlmData : tyUIAllAlm;
END_VAR
(**)
(*Local Output*)
VAR
	eStartupAct : eStartupAction;
	eSimuAct : eSimulationsAction;
	eHWInfoAct : eHWInfoAction;
	eTLBuzAct : eTLBuzAction;
	eRstErrAct : eRstErrAction;
	eProdRcpAct : eProdRcpAction;
	eMpProdRcpAct : eMpProdRcpAction;
	eMagRcpAct1 : eMagRcpAction;
	eMagRcpAct : eMagRcpAction;
	eMcParamAct : eMcParamAction;
	eUsrMgmtAct : eUsrMgmtAction;
	eBuffer1Act : eBufferAction;
	eBuffer2Act : eBufferAction;
	eBuffer3Act : eBufferAction;
	eBuffer4Act : eBufferAction;
	eDSSMEMAAAct : eSMEMAAction;
	eDSSMEMABAct : eSMEMAAction;
	eInShutterAct : ePneuAction;
	eInShutterAct2 : ePneuAction;
	eInShutterAct3 : ePneuAction;
	eOutShutterAct : ePneuAction;
	eOutShutterAct2 : ePneuAction;
	ePullerAct : ePneuAction;
	ePullConvAct : eConvAction;
	eMtrPshrAct : eMtrPshrAction;
	eMagConvSelClp1Act : ePneuAction;
	eMagConvSelClp2Act : ePneuAction;
	eMagConvSelClp3Act : ePneuAction;
	eMagConvSelClp4Act : ePneuAction;
	eMagConv2Clp1Act : eMagConv2ClpAction;
	eMagConv2Clp2Act : eMagConv2ClpAction;
	eMagConv2Clp3Act : eMagConv2ClpAction;
	eMagConv2Clp4Act : eMagConv2ClpAction;
	eAWPushOrPullerAct : eAWAction;
	eAWOpenAct : eAWAction;
	eLifterBtmAct : eLifterAction;
	eTravAct : eTravAction;
	eServoPullPusherAct : ePullerPusherAction;
	eDOAct : eDOAction;
	eHermesAct : eHermesAction;
	eLFLeaderAct : eLFAction;
	eOpsAct : eOperationsAction;
	eUSBRdrAct : eUSBRdrAction;
	eFrmAct : eFrmAction;
	eMag1SafetyBarAct : ePneuAction;
	eMag2SafetyBarAct : ePneuAction;
	eMag3SafetyBarAct : ePneuAction;
	eTrolleyLckAct1 : ePneuAction;
	eTrolleyLckAct2 : ePneuAction;
END_VAR
(*Simu*)
VAR
	eNtWr : eNtParamAction;
	fbSDOWriteAccT : CANopenSDOWrite8;
	fbSDOWriteAccL : CANopenSDOWrite8;
	sDevice : STRING[3] := 'IF7';
	udiAcc : UDINT := 500;
	usiWrStep : USINT;
END_VAR
(**)
VAR
	tyMcParamWr : tyMcParam;
	tyProdRcpInfoIn : tyProdRcpParam;
	sProdRcpSearch : STRING[30];
	sProdRcpScan : STRING[30];
	tyProdRcpCurrRcpWr : tyProdRcpParam;
	tyMagRcpInfoIn : tyMagRcpParam;
	sMagRcpSearch : STRING[30];
	tyMagRcpCurrRcpWr : tyMagRcpParam;
	tyMagRcpInfoIn1 : tyMagRcpParam;
	sMagRcpSearch1 : STRING[30];
	tyMagRcpCurrRcpWr1 : tyMagRcpParam;
	tyUsrMgmtInfoIn : tyUsrMgmtParam;
	tyUsrMgmtAccessRightLvl1Wr : tyUsrMgmtAccessRight;
	tyUsrMgmtAccessRightLvl2Wr : tyUsrMgmtAccessRight;
	tyUsrMgmtAccessRightLvl3Wr : tyUsrMgmtAccessRight;
	a_tyHermesDSParamWr : ARRAY[0..c_diHermesConfigMaxIdx] OF tyHermesDSParam;
	tyHermesSvyParamWr : tyHermesSvyParam;
	sSetIPAddr : STRING[30];
	sSetSubnetMask : STRING[30];
	bManualMod : BOOL := FALSE;
	bUIManualMod : BOOL;
	bMuteBuz : BOOL := FALSE;
	diMnlMtrPshrExtSpd : DINT;
	diMnlMtrPshrExtTorq : DINT;
	diMnlServoMtrMaxPulRatio : DINT := 3000;
	diMnlAWPushOrPullerGoWidth : DINT;
	diMnlAWPushOrPullerNomSpd : DINT;
	diMnlAWPushOrPullerTargetPos : DINT;
	diMnlAWPushOrPullerStepSize : DINT;
	diMnlAWPushOrPullerJogSpd : DINT;
	diMnlAWGoWidth : DINT;
	diMnlAWTargetPos : DINT;
	diMnlAWStepSize : DINT;
	diMnlAWNomSpd : DINT;
	diMnlAWJogSpd : DINT;
	diMnlLifterGoSlt1Pos : DINT;
	diMnlLifterMag1GoSlt : DINT;
	diMnlLifterMag2GoSlt : DINT;
	diMnlLifterMag3GoSlt : DINT;
	diMnlLifterMag4GoSlt : DINT;
	diMnlLifterTargetPos : DINT;
	diMnlLifterStepSize : DINT;
	diMnlLifterNomSpd : DINT;
	diMnlLifterJogSpd : DINT;
	diMnlTravTargetPos : DINT;
	diMnlTravStepSize : DINT;
	diMnlTravNomSpd : DINT;
	diMnlTravJogSpd : DINT;
	bVSMEMADSAEn : BOOL;
	bVSMEMADSBEn : BOOL;
	bVSMEMADSBA : BOOL;
	bVSMEMADSBB : BOOL;
	bLeaderRun : BOOL;
	bProdAccData : BOOL;
	bOpsBypsInitConv : BOOL;
	bAIVCommReconnect : BOOL;
	bNewMag1 : BOOL;
	bNewMag2 : BOOL;
	bNewMag3 : BOOL;
	bNewMag4 : BOOL;
	bRlsMag1 : BOOL;
	bRlsMag2 : BOOL;
	bRlsMag3 : BOOL;
	bRlsMag4 : BOOL;
	bEjectMag1 : BOOL;
	bEjectMag2 : BOOL;
	bEjectMag3 : BOOL;
	tyAGVSimulateSig : tyTagAGVToDTMag;
	bAGVSimulateOnline : BOOL;
	bAGVSimulationOn : BOOL;
	bUnloadMag : BOOL;
	fbUnloadBlinkTm : TON := (PT:=T#500ms);
	diMnlPPGoWidth : DINT;
	diMnlPPTargetPos : DINT;
	diMnlPPStepSize : DINT;
	diMnlPPNomSpd : DINT;
	diMnlPPJogSpd : DINT;
END_VAR
VAR RETAIN
	bHCommModChg : BOOL;
END_VAR
(**)
(*Local Input*)
(**)
(*Local*)
VAR
	bInitDone : BOOL := FALSE;
	bInitialDone : BOOL;
	eUIInit : eUIInitial := UIInitialC0005;
	i : UINT := 0;
	eChgPage : ePage := UIP0001Startup;
	eChgPageOld : ePage := UIP0001Startup;
	eCurrPage : ePage := UIP0001Startup;
	bChgPage : BOOL;
	bJogFast : BOOL := FALSE;
	bJogSlow : BOOL := FALSE;
	bJogStopAWPushOrPuller : BOOL := FALSE;
	bJogStopAW : BOOL := FALSE;
	bJogStopTrav : BOOL := FALSE;
	bJogStopLifter : BOOL := FALSE;
	bLoginSuccess : BOOL := FALSE;
	bRefreshMagRcpDetail : BOOL := FALSE;
	bRefreshMagRcpTable1 : BOOL := TRUE;
	bRefreshMagRcpTable : BOOL := TRUE;
	bRefreshProdRcpDetail : BOOL := FALSE;
	bRefreshProdRcpTable : BOOL := TRUE;
	bRefreshUsrMgmtTable : BOOL := TRUE;
	bMagazineRcpA : BOOL := TRUE;
	bMagazineRcpB : BOOL := TRUE;
	bTeachTravPosA : BOOL := FALSE;
	bTeachTravPosB : BOOL := FALSE;
	bTeachLifterPosA : BOOL := FALSE;
	bTeachLifterPosB : BOOL := FALSE;
	bTeachLifterMag1Slt1Pos : BOOL := FALSE;
	bTeachLifterMag2Slt1Pos : BOOL := FALSE;
	bTeachLifterMag3Slt1Pos : BOOL := FALSE;
	bTeachLifterMag4Slt1Pos : BOOL := FALSE;
	bTeachTravPosMag1 : BOOL := FALSE;
	bTeachTravPosMag2 : BOOL := FALSE;
	bTeachTravPosMag3 : BOOL := FALSE;
	bTeachTravPosMag4 : BOOL := FALSE;
	usiTestTravStep : USINT := 0;
	bOnlineTemp : BOOL := FALSE;
	bIPDuplicate : BOOL := FALSE;
	usiLoginStep : USINT := 0;
	usiSelProdRcpStep : USINT := 0;
	usiSelMagRcpStep1 : USINT := 0;
	usiSelMagRcpStep : USINT := 0;
	usiSaveCommStep : USINT := 0;
	usiSaveAIVCommStep : USINT := 0;
	usiSaveSubnetMaskStep : USINT := 0;
	usiSaveIPAddrStep : USINT := 0;
	usiSaveUsrMgmtStep : USINT := 0;
	usiEditUsrMgmtStep : USINT := 0;
	usiDelUsrMgmtStep : USINT := 0;
	usiSaveProdRcpStep : USINT := 0;
	usiDelProdRcpStep : USINT := 0;
	usiProdRcpToXMLStep : USINT := 0;
	usiProdRcpFromXMLStep : USINT := 0;
	usiSaveMagRcpStep : USINT := 0;
	usiDelMagRcpStep : USINT := 0;
	usiChgPage : USINT := 1;
	usiLFLeaderCtrlStep : USINT := 0;
	usiDelMcDetailsStep : USINT := 0;
	usiTableShftStep : USINT := 0;
	usiSimuMod : USINT := 0;
	usiSimuNtStep : USINT := 0;
	usiNetworkModeSelected : USINT;
	fbShutterSimChgOver : TON := (PT:=T#1500ms);
	fbActSimuTmr : TON;
	fbSSaverTm : TON := (0);
	fbJogSlowToFastDlyTm : TON := (IN:=FALSE,PT:=T#2s,Q:=FALSE,ET:=0,StartTime:=0,M:=FALSE,Restart:=0);
	fbLmtRstTm : TON := (PT:=T#1s);
	fbErrBlinkTm : TON := (IN:=FALSE,PT:=T#1s,Q:=FALSE,ET:=0,StartTime:=0,M:=FALSE,Restart:=0);
	fbRstBlinkTm : TON := (IN:=FALSE,PT:=T#1s,Q:=FALSE,ET:=0,StartTime:=0,M:=FALSE,Restart:=0);
	fbAccDatBlinkTm : TON := (IN:=FALSE,PT:=T#500ms,Q:=FALSE,ET:=0,StartTime:=0,M:=FALSE,Restart:=0);
	fbBypsInitConvBlinkTm : TON := (PT:=T#500ms);
	fbMcStatUpdtTm : TON := (IN:=FALSE,PT:=T#1s,Q:=FALSE,ET:=0,StartTime:=0,M:=FALSE,Restart:=0);
	fbStopBlinkTm : TON := (IN:=FALSE,PT:=T#500ms,Q:=FALSE,ET:=0,StartTime:=0,M:=FALSE,Restart:=0);
	fbLFLeaderCtrlBlinkTm : TON := (IN:=FALSE,PT:=T#500ms,Q:=FALSE,ET:=0,StartTime:=0,M:=FALSE,Restart:=0);
	fbMag1EntrySenOnTm : TON := (PT:=T#3s);
	fbMag2EntrySenOnTm : TON := (PT:=T#3s);
	fbMag3EntrySenOnTm : TON := (PT:=T#3s);
	tyP0400Table : tyTable := (bSliderActive:=FALSE,bTableActive:=FALSE,sVisuNm:='Visu',uiSelectedRow:=1,uiSelectedRowOld:=1,uiTablePos:=1);
	fbP0400Table : fbTableCtrl;
	tyP0410Table : tyTable := (bSliderActive:=FALSE,bTableActive:=FALSE,sVisuNm:='Visu',uiSelectedRow:=1,uiSelectedRowOld:=1,uiTablePos:=1);
	tyP0410Table1 : tyTable := (bSliderActive:=FALSE,bTableActive:=FALSE,sVisuNm:='Visu',uiSelectedRow:=1,uiSelectedRowOld:=1,uiTablePos:=1);
	fbP0410Table : fbTableCtrl;
	fbP0410Table1 : fbTableCtrl;
	tyP0700Table : tyTable := (bSliderActive:=FALSE,bTableActive:=FALSE,sVisuNm:='Visu',uiSelectedRow:=1,uiSelectedRowOld:=1,uiTablePos:=1);
	fbP0700Table : fbTableCtrl;
	tyP0800Table1 : tyTable := (bSliderActive:=FALSE,bTableActive:=FALSE,sVisuNm:='Visu',uiSelectedRow:=1,uiSelectedRowOld:=1,uiTablePos:=1);
	fbP0800Table1 : fbTableCtrl;
	tyP0800Table2 : tyTable := (bSliderActive:=FALSE,bTableActive:=FALSE,sVisuNm:='Visu',uiSelectedRow:=1,uiSelectedRowOld:=1,uiTablePos:=1);
	fbP0800Table2 : fbTableCtrl;
	tyP0800Table3 : tyTable := (bSliderActive:=FALSE,bTableActive:=FALSE,sVisuNm:='Visu',uiSelectedRow:=1,uiSelectedRowOld:=1,uiTablePos:=1);
	fbP0800Table3 : fbTableCtrl;
	tyP0800Table4 : tyTable := (bSliderActive:=FALSE,bTableActive:=FALSE,sVisuNm:='Visu',uiSelectedRow:=1,uiSelectedRowOld:=1,uiTablePos:=1);
	fbP0800Table4 : fbTableCtrl;
	tyP1030Table : tyTable := (bSliderActive:=FALSE,bTableActive:=FALSE,sVisuNm:='Visu',uiSelectedRow:=1,uiSelectedRowOld:=1,uiTablePos:=1);
	fbP1030Table : fbTableCtrl_v2;
	tyP1040Table : tyTable := (bSliderActive:=FALSE,bTableActive:=FALSE,sVisuNm:='Visu',uiSelectedRow:=1,uiSelectedRowOld:=1,uiTablePos:=1);
	fbP1040Table : fbTableCtrl_v2;
	tyP1050Table : tyTable := (bSliderActive:=FALSE,bTableActive:=FALSE,sVisuNm:='Visu',uiSelectedRow:=1,uiSelectedRowOld:=1,uiTablePos:=1);
	fbP1050Table : fbTableCtrl;
	tyP1080Table : tyTable := (bSliderActive:=FALSE,bTableActive:=FALSE,sVisuNm:='Visu',uiSelectedRow:=1,uiSelectedRowOld:=1,uiTablePos:=1);
	fbP1080Table : fbTableCtrl;
	udiP1030SelectedRowOld : UDINT := 0;
	udiP1030SelectedRow : UDINT := 0;
	udiP1040SelectedRowOld : UDINT := 0;
	udiP1040SelectedRow : UDINT := 0;
	usiP1080SelectedLvl : USINT := 0;
	udiP1080SelectedRow : UDINT := 0;
	uiSSaverCnt : UINT := 0;
	a_iIPPart1 : ARRAY[1..4] OF INT := [4(0)];
	a_iIPPart2 : ARRAY[1..4] OF INT := [4(0)];
	a_iSubnetMaskPart1 : ARRAY[1..4] OF INT := [4(0)];
	sLFIPAddrTemp : STRING[15];
	bCheckDone : BOOL;
	bFilterSortP0400 : BOOL;
	bFilterSortP1040 : BOOL;
	iSelectedRowValue : UINT;
	bUpdateP0400Table : BOOL;
	bUpdateP0410Table1 : BOOL;
	bUpdateP0410Table : BOOL;
	bUpdateP1030Table : BOOL;
	bUpdateP1040Table : BOOL;
	bUpdateP1030LoadData : BOOL;
	bUpdateP1040LoadData : BOOL;
	bChgPageDone : BOOL; (*Auto Logout*)
	bMismatchOverWriteConfig : BOOL;
	bTempAddrFillDone : BOOL;
	sTempIPAddr : STRING[15];
	sTempSubnetMask : STRING[15];
	bIPConfigChgDone : BOOL;
	bOverwriteIP : BOOL;
	bOverwriteSubnet : BOOL;
	bOverwriteEthMode : BOOL;
	bSaveNetworkPriority : BOOL;
	bNetworkConfigChanged : BOOL;
	bTeachServo : BOOL := FALSE;
	usiNetworkModeOld : USINT;
	usiNetworkModeNew : USINT;
	usiChgNetworkConfigStep : USINT := 0;
	usiRefreshDetailStep : USINT := 0;
END_VAR
(*AutoLogout*)
VAR
	bPromptSessionExp : BOOL := FALSE;
	fbAutoLogoutTm : TON;
	fbTouchTm : fbTouchGetAction := (sVisuNm:='Visu');
END_VAR
(*LF*)
VAR
	bLFRunInBG : BOOL;
	bLFDeleteOn : BOOL;
	bUpdateP1050Table : BOOL;
	iIPExtract : INT;
	sLFSettingCurrentIP : STRING[4];
	iLFSettingCurrentIP : INT;
	sLFSettingAutoFill : STRING[15];
	sLFSettingTemp : STRING[15];
	bLFSettingAutoFill : BOOL;
	bLFSettingAutoClear : BOOL;
END_VAR
(*Network*)
VAR
	udiTempEthMode : UDINT;
	bUpdateP1021Network : BOOL;
	uiLFStartEditNo : UINT;
	tySOTSimulateSig1 : tyLyrP0950SOTstatus;
	tySOTSimulateSig2 : tyLyrP0950SOTstatus;
	tySOTSimulateSig3 : tyLyrP0950SOTstatus;
	tySOTSimulateSig4 : tyLyrP0950SOTstatus;
END_VAR
(*AIV COMM*)
VAR
	bSOTMagErr1 : BOOL := FALSE;
	bSOTMagErr2 : BOOL := FALSE;
	bSOTMagErr3 : BOOL := FALSE;
	bSOTMagErr4 : BOOL := FALSE;
	bSOTMagRdy1 : BOOL := FALSE;
	bSOTMagRdy2 : BOOL := FALSE;
	bSOTMagRdy3 : BOOL := FALSE;
	bSOTMagRdy4 : BOOL := FALSE;
	bSOTMagAvail1 : BOOL := FALSE;
	bSOTMagAvail2 : BOOL := FALSE;
	bSOTMagAvail3 : BOOL := FALSE;
	bSOTMagAvail4 : BOOL := FALSE;
	bSOTMagSLarge1 : BOOL := FALSE;
	bSOTMagSLarge2 : BOOL := FALSE;
	bSOTMagSLarge3 : BOOL := FALSE;
	bSOTMagSLarge4 : BOOL := FALSE;
	bDisplayMag4Info : BOOL := FALSE;
	bAIVReqBring1 : BOOL := FALSE;
	bAIVReqBring2 : BOOL := FALSE;
	bAIVReqBring3 : BOOL := FALSE;
	bAIVReqBring4 : BOOL := FALSE;
	bAIVReqGet1 : BOOL := FALSE;
	bAIVReqGet2 : BOOL := FALSE;
	bAIVReqGet3 : BOOL := FALSE;
	bAIVReqGet4 : BOOL := FALSE;
END_VAR
(*MagConv*)
VAR
	bDispMagConv1 : BOOL := TRUE;
	bDispMagConv2 : BOOL := FALSE;
	bDispMagConv3 : BOOL := FALSE;
	bDispMagConv4 : BOOL := FALSE;
END_VAR
(*USB Barcode Scanner*)
VAR
	usiChgRcpStep : USINT;
	usiUSBBarcodeStep : USINT;
	bUSBRun : BOOL;
	bResetButton : BOOL;
	bErrorled : BOOL;
	bUSBConnecting : BOOL;
	bUSBClose : BOOL;
	bManualEntry : BOOL;
	strcmp_status : DINT := 0;
	sUSBBarcode : STRING[255] := '';
	bUSBDisconnected : BOOL;
	bWorkOrderDisp : BOOL := TRUE;
END_VAR
(**)
VAR
	bDispSafetyBar1 : BOOL := TRUE;
	bDispSafetyBar2 : BOOL := FALSE;
	bDispSafetyBar3 : BOOL := FALSE;
END_VAR
(**)
(*opcUA to LMC*)
VAR RETAIN
	tyTagNm : tyUITagNm;
	uiBrdOutCntr : UINT;
END_VAR
VAR
	bInitQuanValue : BOOL;
	bMag1Active : BOOL;
	bMag2Active : BOOL;
	fbLMCfbTm : TON;
	diMag1TtSlt : DINT;
	diMag2TtSlt : DINT;
	diTtWorkOrderSlt : DINT;
	string1 : STRING[80];
	string2 : STRING[80];
END_VAR
(*Output*)
VAR
	bBlkOpsTravLif : BOOL;
	bSafetyCurtainReset : BOOL;
	bBypCurtainSen : BOOL;
	bBypCurtainPBLED : BOOL;
	fbCurtainRstDly : TON := (PT:=T#500ms);
	bMachineSafetySigToDS : BOOL;
END_VAR
(**)
(*Start Hermes var*)
VAR
	bNaviLyr1 : BOOL;
	bNaviLyr2 : BOOL;
	bQueryBoardInfo : BOOL := FALSE;
	bQueryWorkOrderInfo : BOOL := FALSE;
	bDeleteWorkOrder : BOOL := FALSE;
	bSaveHMISvyConfig : BOOL;
	bSaveHMIConfigure : BOOL;
	bSkipWorkOrder : BOOL;
	bReadWorkOrder : BOOL;
	iSlotId : INT := 0;
END_VAR
(*end Hermes var*)
```
